FUNCTION_BLOCK FB_Example
CONST
    MAX_LEN := 10;
END_CONST
VAR
    x : INT;
END_VAR
BEGIN
x := MAX_LEN;
END_FUNCTION_BLOCK
